PROGRAM PRG_ADS_Interfaces
VAR
	
	counter_x : INT;
   //Reading from LAMP PLC

	// This variable needs to be instantiated for the Watchdog to work
	i_iWatchdog : UDINT;
	
	// create watch dog for LAMP PLC
	ads_watch_dog : FB_ADS_WATCHDOG;
	
END_VAR



lamp_turbo_running_reader(
	sNetId := '172.21.132.34.1.1', // AMS NET ID of PLC being read from
	nPort := 851, // ADS port of the PLC reading from this PLC
	sVarName := 'Main.b_PumpRunning', // Full name of the FB containing the gauge to be read
	iWatchdog := i_iWatchdog // UDINT required for watchdog functionality
);


LAMP_ROUGH_GPI02_reader(
	sNetId := '172.21.132.34.1.1', // AMS NET ID of PLC being read from
	nPort := 851, // ADS port of the PLC reading from this PLC
	sVarName := 'GVL_Devices.LAMP_ROUGH_GPI_02', // Full name of the FB containing the gauge to be read
	iWatchdog := i_iWatchdog // UDINT required for watchdog functionality
);

LAMP_ROUGH_GPI04_reader(
	sNetId := '172.21.132.34.1.1', // AMS NET ID of PLC being read from
	nPort := 851, // ADS port of the PLC reading from this PLC
	sVarName := 'GVL_Devices.LAMP_ROUGH_GPI_04', // Full name of the FB containing the gauge to be read
	iWatchdog := i_iWatchdog // UDINT required for watchdog functionality
);


ads_watch_dog(
	sNetId := '172.21.132.34.1.1', // AMS NET ID of LAMP PLC reading from this PLC
	nPort := 851, // ADS port of the PLC reading from this PLC
	sVarName := 'Main.i_iWatchdog', // Full name of the UDINT provided to the 'iWatchdog' parameter in the interface functions on the PLC reading from this PLC 
);

END_PROGRAM

(* stored: Version 1.1.0.1, ProductVersion 3.1.4022.18
   POU PRG_ADS_Interfaces: Id {a2c26feb-aa2b-4b7d-a0d4-a5da6570030a}, SpecialFunc None *)
